{attribute 'qualified_only'}
{attribute 'strict'}
TYPE E_FatalErrors :
(
    NO_FATAL_ERROR := 0,
    NoStopDetectedSynch := 20,
    ValveBlockedSynch := 21,
    ValveBlocked := 22,
    StepLossSynch := 25,
    MotorDriverFault := 40
) UINT := NO_FATAL_ERROR;
END_TYPE

(* stored: Version 1.1.0.1
   DUT E_FatalErrors: Id {a7468a7d-d8ef-44f4-83de-890c933bd59d} *)
